# EPICS substitutions: iocBoot/iocJenaNV100D/JenaNV100D.substitutions
file "$(TOP)/db/JenaNV100D.template"
{
pattern
{P,         C,      PORT}
{IOC:, jena1:, serial1}
}

file "$(STD)/stdApp/Db/genTweak.db"
{
pattern
{P,       N, PREC,           PV}
{IOC:, jena1:, 3, IOC:jena1:write}
}
